{attribute 'linkalways'} 
{attribute 'no_explicit_call' := 'This FB is a CLASS and must be accessed using methods or properties'}
{attribute 'enable_dynamic_creation'}
FUNCTION_BLOCK FINAL LE_ULINT EXTENDS Node
VAR
	in1 : _ULINT(0);
	in2 : _ULINT(0);
	out : _BOOL(FALSE);
END_VAR

METHOD PUBLIC Clone : I_Node
VAR
	pNode : POINTER TO LE_ULINT;
END_VAR
pNode := __NEW(LE_ULINT);
Clone := pNode^;
END_METHOD

METHOD FB_init : BOOL
VAR_INPUT
	bInitRetains : BOOL; // if TRUE, the retain variables are initialized (warm start / cold start)
	bInCopyCode : BOOL;  // if TRUE, the instance afterwards gets moved into the copy code (online change)
END_VAR
AddInput('in1',THIS^.in1);
AddInput('in2',THIS^.in2);
AddOutput('out', THIS^.out);
END_METHOD

METHOD PROTECTED OnExecute
VAR
END_VAR
out.Value := in1.Value <= in2.Value;
END_METHOD

END_FUNCTION_BLOCK

(* stored: Version 1.1.0.1, ProductVersion 3.1.4024.15
   POU LE_ULINT: Id {9a9a9e58-e2e3-4138-9b92-906c01b82319}, SpecialFunc None
   Folder Constructor: Id {2fc7f464-0fab-4446-a1a7-79967872488d}
   Method Clone: Id {9397cdad-54ef-40d8-bc4d-6559dbc7d674}
   Method FB_init: Id {97f2a623-830c-4285-8c0f-97d36800c7af}
   Method OnExecute: Id {ad73dffe-e143-4836-b0dc-f3da17c8b4ad} *)
